TYPE EL3154_CHANNEL :
	STRUCT
		
	
	Status 	AT %I* : EL3154_DEV_STATUS;
	Value 	AT %I* : INT;
	
	
	END_STRUCT
END_TYPE

(* stored: Version 1.1.0.1, ProductVersion 3.1.4024.15
   DUT EL3154_CHANNEL: Id {c4550133-d8e3-40dd-88c9-eedd7ad1fa4b} *)
